// TIA Portal V16 export
// export: Created 2023-01-04T15:44:08.7039058Z, ExportSetting WithDefaults, DisplayName Totally Integrated Automation Portal, DisplayVersion V16, DisplayName TIA Portal Version Control Interface, DisplayVersion V16, DisplayName TIA Portal Openness, DisplayVersion V16, DisplayName STEP 7 Professional, DisplayVersion V16, DisplayName STEP 7 Safety, DisplayVersion V16, DisplayName WinCC Advanced, DisplayVersion V16
FUNCTION_BLOCK "Filling_Logic"   // FB2, LAD
{ S7_Optimized_Access := 'TRUE' }
VERSION : 0.1
// stored: AutoNumber true, IsIECCheckEnabled false, IsRetainMemResEnabled false, MemoryReserve 100, SetENOAutomatically false, UDAEnableTagReadback false
   VAR_INPUT
      PS2_Filling_Station : Bool;
      FIC_B102 : Int;
      Liquid_AorB_in_Bottle_ml : Real;
      Liquid_AorB_pct : Int;
      PTRIG3 : Bool;
      PTRIG2 : Bool;
      Wait_to_fill : Time;
   END_VAR
   VAR_OUTPUT
      Outlet_of_tanks : Bool;
      Flow_ml_per_sec : Real;
      PTRIG1 : Bool;
      FillingData_LiqAorB_ml : Real;
   END_VAR
BEGIN

REGION Network 1
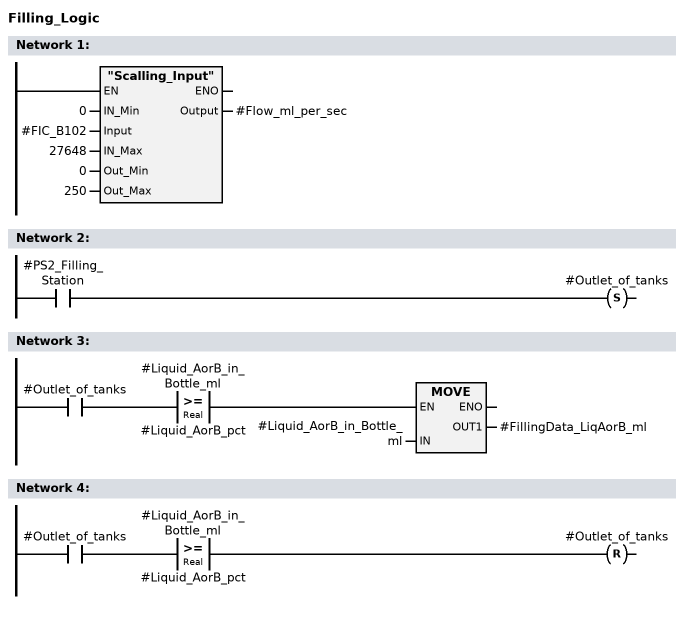
   RUNG wire#powerrail
      "Scalling_Input"(IN_Min := 0, Input := #FIC_B102, IN_Max := 27648, Out_Min := 0, Out_Max := 250, Output => #Flow_ml_per_sec)
   END_RUNG
   // the same network as SCL:
   "Scalling_Input"(IN_Min := 0,
                    Input := #FIC_B102,
                    IN_Max := 27648,
                    Out_Min := 0,
                    Out_Max := 250,
                    Output => #Flow_ml_per_sec);
END_REGION

REGION Network 2
   RUNG wire#powerrail
      Contact( #PS2_Filling_Station )
      S_Coil( #Outlet_of_tanks )
   END_RUNG
   // the same network as SCL:
   IF #PS2_Filling_Station THEN #Outlet_of_tanks := TRUE; END_IF;
END_REGION

REGION Network 3
   RUNG wire#powerrail
      Contact( #Outlet_of_tanks )
      { S7_Templates := "SrcType := Real" } GE_Contact(in1 := #Liquid_AorB_in_Bottle_ml, in2 := #Liquid_AorB_pct)
      Move(in := #Liquid_AorB_in_Bottle_ml, out1 => #FillingData_LiqAorB_ml)
   END_RUNG
   // the same network as SCL:
   IF #Outlet_of_tanks AND (#Liquid_AorB_in_Bottle_ml >= #Liquid_AorB_pct) THEN
       #FillingData_LiqAorB_ml := #Liquid_AorB_in_Bottle_ml;
   END_IF;
END_REGION

REGION Network 4
   RUNG wire#powerrail
      Contact( #Outlet_of_tanks )
      { S7_Templates := "SrcType := Real" } GE_Contact(in1 := #Liquid_AorB_in_Bottle_ml, in2 := #Liquid_AorB_pct)
      R_Coil( #Outlet_of_tanks )
   END_RUNG
   // the same network as SCL:
   IF #Outlet_of_tanks AND (#Liquid_AorB_in_Bottle_ml >= #Liquid_AorB_pct) THEN
       #Outlet_of_tanks := FALSE;
   END_IF;
END_REGION
END_FUNCTION_BLOCK
